% RSLogix 500 project PROJECT4_MULTIPOSITION_SERVO.RSS, saved by version 8.30.00.16 %
PROJECT "UNTITLED"    % processor: Bul.1763 MicroLogix 1100 Series B %

PROGRAM FILES
  LAD 2 "MAIN"  3 rungs
  LAD 3 "I/O"  8 rungs
  LAD 4 "CONTROL"  18 rungs

DATA FILES
  O0 OUTPUT  4 elements
  I1 INPUT  6 elements
  S2 STATUS  66 elements
  B3 BINARY  2 elements
  T4 TIMER  3 elements
  C5 COUNTER  1 elements
  R6 CONTROL  1 elements
  N7 INTEGER  1 elements
  F8 FLOAT  1 elements

LADDER 2 "MAIN"
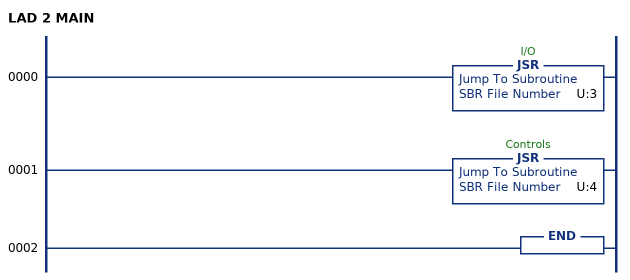
% Rung: 0 %
SOR JSR U:3 EOR
%   U:3  "I/O" %
% Rung: 1 %
SOR JSR U:4 EOR
%   U:4  "Controls" %
% Rung: 2 %
SOR END EOR

LADDER 3 "I/O"
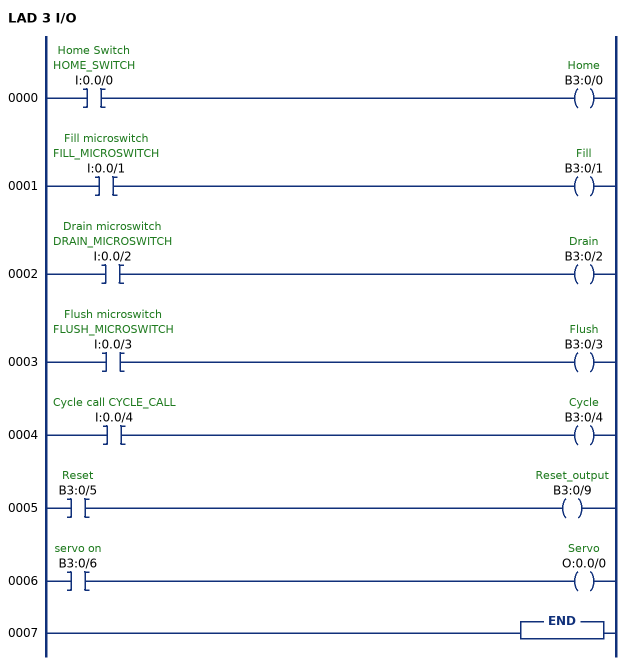
% Rung: 0 %
SOR XIC I:0.0/0 OTE B3:0/0 EOR
%   I:0.0/0  HOME_SWITCH  "Home Switch" %
%   B3:0/0  "Home" %
% Rung: 1 %
SOR XIC I:0.0/1 OTE B3:0/1 EOR
%   I:0.0/1  FILL_MICROSWITCH  "Fill microswitch" %
%   B3:0/1  "Fill" %
% Rung: 2 %
SOR XIC I:0.0/2 OTE B3:0/2 EOR
%   I:0.0/2  DRAIN_MICROSWITCH  "Drain microswitch" %
%   B3:0/2  "Drain" %
% Rung: 3 %
SOR XIC I:0.0/3 OTE B3:0/3 EOR
%   I:0.0/3  FLUSH_MICROSWITCH  "Flush microswitch" %
%   B3:0/3  "Flush" %
% Rung: 4 %
SOR XIC I:0.0/4 OTE B3:0/4 EOR
%   I:0.0/4  CYCLE_CALL  "Cycle call" %
%   B3:0/4  "Cycle" %
% Rung: 5 %
SOR XIC B3:0/5 OTE B3:0/9 EOR
%   B3:0/5  "Reset" %
%   B3:0/9  "Reset_output" %
% Rung: 6 %
SOR XIC B3:0/6 OTE O:0.0/0 EOR
%   B3:0/6  "servo on" %
%   O:0.0/0  "Servo" %
% Rung: 7 %
SOR END EOR

LADDER 4 "CONTROL"
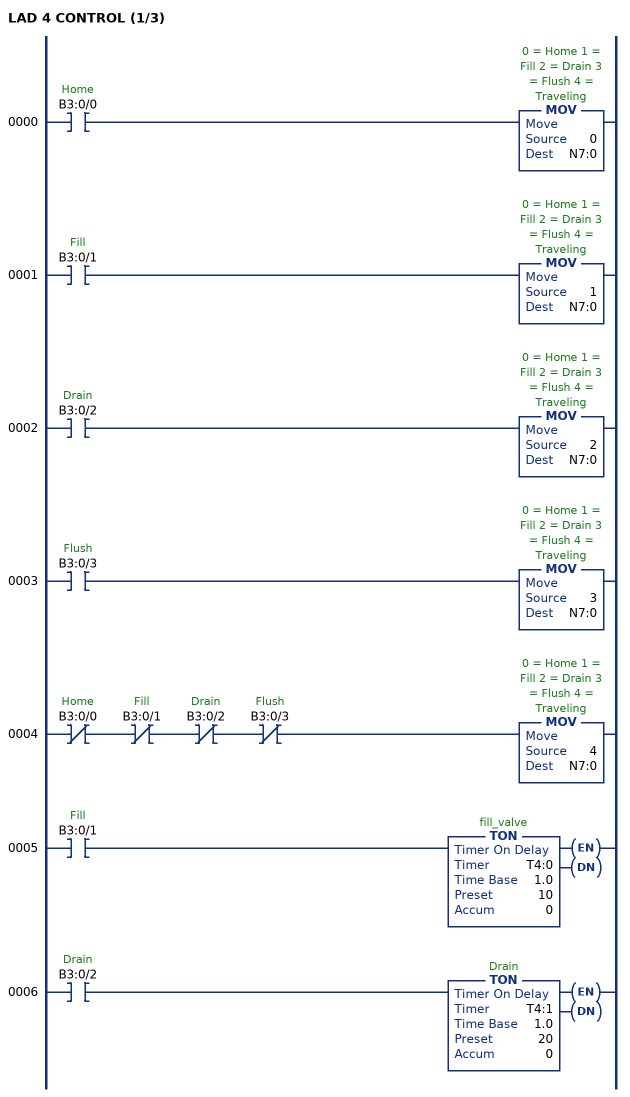
% Rung: 0 %
SOR XIC B3:0/0 MOV 0 N7:0 EOR
%   B3:0/0  "Home" %
%   N7:0  "0 = Home 1 = Fill 2 = Drain 3 = Flush 4 = Traveling" %
% Rung: 1 %
SOR XIC B3:0/1 MOV 1 N7:0 EOR
%   B3:0/1  "Fill" %
%   N7:0  "0 = Home 1 = Fill 2 = Drain 3 = Flush 4 = Traveling" %
% Rung: 2 %
SOR XIC B3:0/2 MOV 2 N7:0 EOR
%   B3:0/2  "Drain" %
%   N7:0  "0 = Home 1 = Fill 2 = Drain 3 = Flush 4 = Traveling" %
% Rung: 3 %
SOR XIC B3:0/3 MOV 3 N7:0 EOR
%   B3:0/3  "Flush" %
%   N7:0  "0 = Home 1 = Fill 2 = Drain 3 = Flush 4 = Traveling" %
% Rung: 4 %
SOR XIO B3:0/0 XIO B3:0/1 XIO B3:0/2 XIO B3:0/3 MOV 4 N7:0 EOR
%   B3:0/0  "Home" %
%   B3:0/1  "Fill" %
%   B3:0/2  "Drain" %
%   B3:0/3  "Flush" %
%   N7:0  "0 = Home 1 = Fill 2 = Drain 3 = Flush 4 = Traveling" %
% Rung: 5 %
SOR XIC B3:0/1 TON T4:0 1.0 10 0 EOR
%   B3:0/1  "Fill" %
%   T4:0  "fill_valve" %
% Rung: 6 %
SOR XIC B3:0/2 TON T4:1 1.0 20 0 EOR
%   B3:0/2  "Drain" %
%   T4:1  "Drain" %

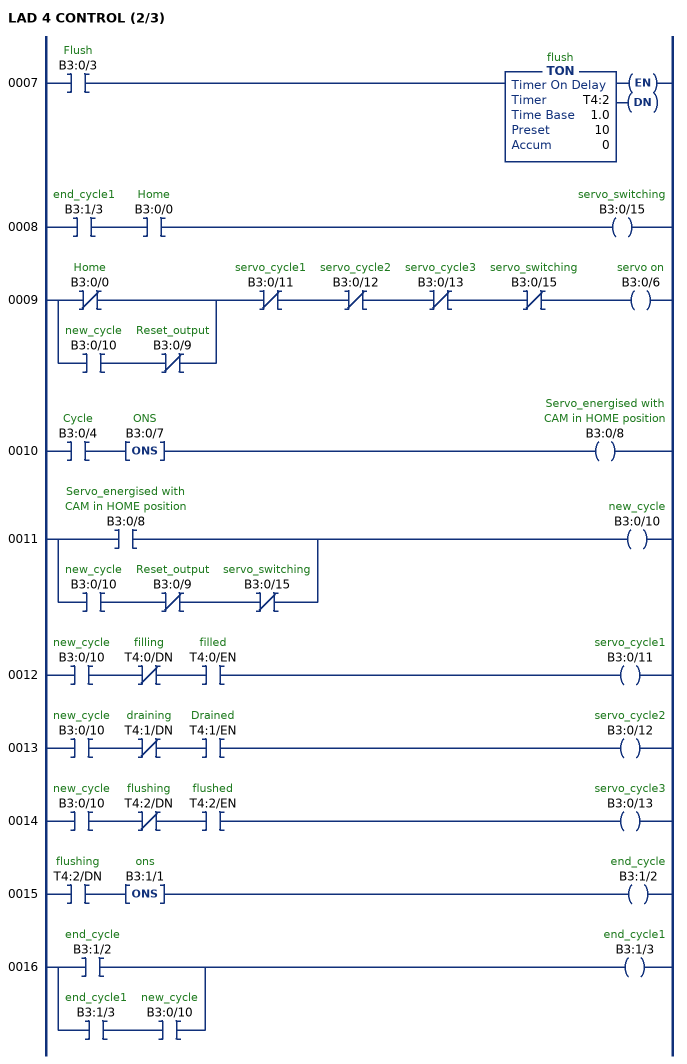
% Rung: 7 %
SOR XIC B3:0/3 TON T4:2 1.0 10 0 EOR
%   B3:0/3  "Flush" %
%   T4:2  "flush" %
% Rung: 8 %
SOR XIC B3:1/3 XIC B3:0/0 OTE B3:0/15 EOR
%   B3:1/3  "end_cycle1" %
%   B3:0/0  "Home" %
%   B3:0/15  "servo_switching" %
% Rung: 9 %
SOR BST XIO B3:0/0 NXB XIC B3:0/10 XIO B3:0/9 BND XIO B3:0/11 XIO B3:0/12 XIO B3:0/13 XIO B3:0/15 OTE B3:0/6 EOR
%   B3:0/0  "Home" %
%   B3:0/10  "new_cycle" %
%   B3:0/9  "Reset_output" %
%   B3:0/11  "servo_cycle1" %
%   B3:0/12  "servo_cycle2" %
%   B3:0/13  "servo_cycle3" %
%   B3:0/15  "servo_switching" %
%   B3:0/6  "servo on" %
% Rung: 10 %
SOR XIC B3:0/4 ONS B3:0/7 OTE B3:0/8 EOR
%   B3:0/4  "Cycle" %
%   B3:0/7  "ONS" %
%   B3:0/8  "Servo_energised with CAM in HOME position" %
% Rung: 11 %
SOR BST XIC B3:0/8 NXB XIC B3:0/10 XIO B3:0/9 XIO B3:0/15 BND OTE B3:0/10 EOR
%   B3:0/8  "Servo_energised with CAM in HOME position" %
%   B3:0/10  "new_cycle" %
%   B3:0/9  "Reset_output" %
%   B3:0/15  "servo_switching" %
% Rung: 12 %
SOR XIC B3:0/10 XIO T4:0/DN XIC T4:0/EN OTE B3:0/11 EOR
%   B3:0/10  "new_cycle" %
%   T4:0/DN  "filling" %
%   T4:0/EN  "filled" %
%   B3:0/11  "servo_cycle1" %
% Rung: 13 %
SOR XIC B3:0/10 XIO T4:1/DN XIC T4:1/EN OTE B3:0/12 EOR
%   B3:0/10  "new_cycle" %
%   T4:1/DN  "draining" %
%   T4:1/EN  "Drained" %
%   B3:0/12  "servo_cycle2" %
% Rung: 14 %
SOR XIC B3:0/10 XIO T4:2/DN XIC T4:2/EN OTE B3:0/13 EOR
%   B3:0/10  "new_cycle" %
%   T4:2/DN  "flushing" %
%   T4:2/EN  "flushed" %
%   B3:0/13  "servo_cycle3" %
% Rung: 15 %
SOR XIC T4:2/DN ONS B3:1/1 OTE B3:1/2 EOR
%   T4:2/DN  "flushing" %
%   B3:1/1  "ons" %
%   B3:1/2  "end_cycle" %
% Rung: 16 %
SOR BST XIC B3:1/2 NXB XIC B3:1/3 XIC B3:0/10 BND OTE B3:1/3 EOR
%   B3:1/2  "end_cycle" %
%   B3:1/3  "end_cycle1" %
%   B3:0/10  "new_cycle" %

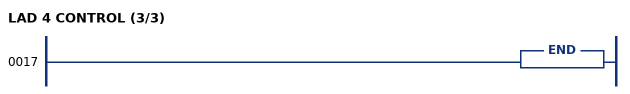
% Rung: 17 %
SOR END EOR

OTHER DOCUMENTED ADDRESSES
  B3:0/14  "ONS"
  B3:1/0  "flushed"

DATA TABLE (non-zero values as saved)
DATA T4
% .PRE .ACC %
% T4:0 % 10 0
% T4:1 % 20 0
% T4:2 % 10 0
